PROGRAM Stn4
VAR

	start4: BOOL;
	reset4: BOOL;

	Stn4ProcessFE: F_TRIG;
	Stn4ProcessRE: R_TRIG;
	bCutStn4ProcessHalt: BOOL;
	DoorClose4: R_TRIG;
	bStn4DoorClamp: BOOL;
END_VAR
VAR // added by the converter: edge detectors and wires of the graphical bodies
    _w1, _w2 : ANY;
END_VAR

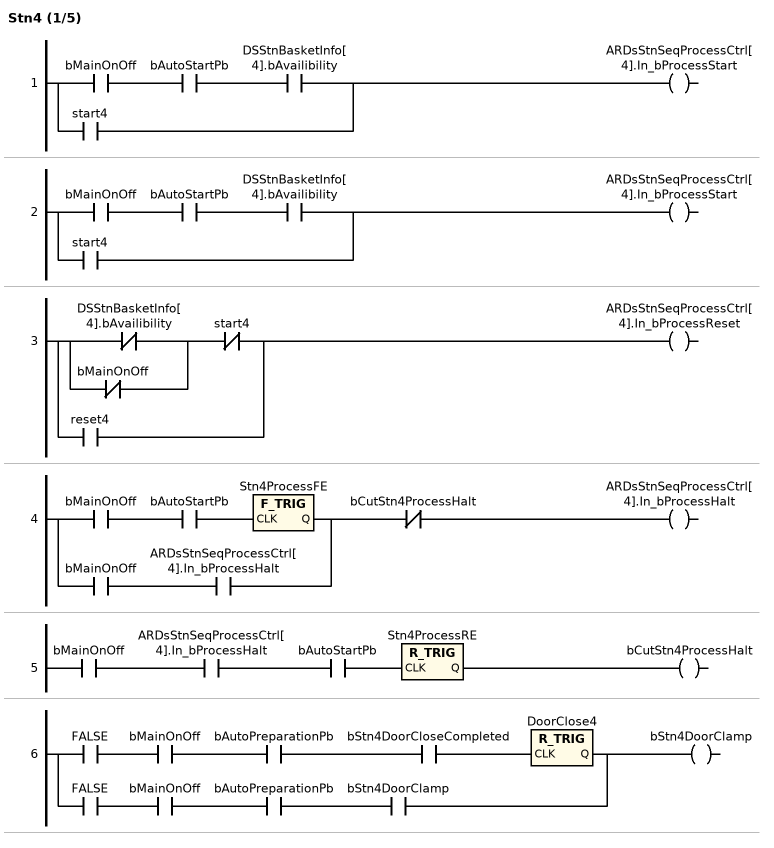
// NETWORK 1
ARDsStnSeqProcessCtrl[4].In_bProcessStart := bMainOnOff AND bAutoStartPb AND DSStnBasketInfo[4].bAvailibility OR start4;

// NETWORK 2
ARDsStnSeqProcessCtrl[4].In_bProcessStart := bMainOnOff AND bAutoStartPb AND DSStnBasketInfo[4].bAvailibility OR start4;

// NETWORK 3
ARDsStnSeqProcessCtrl[4].In_bProcessReset := (NOT DSStnBasketInfo[4].bAvailibility OR NOT bMainOnOff) AND NOT start4 OR reset4;

// NETWORK 4
Stn4ProcessFE(CLK := bMainOnOff AND bAutoStartPb); // F_TRIG
ARDsStnSeqProcessCtrl[4].In_bProcessHalt := (Stn4ProcessFE.Q OR bMainOnOff AND ARDsStnSeqProcessCtrl[4].In_bProcessHalt) AND NOT bCutStn4ProcessHalt;

// NETWORK 5
Stn4ProcessRE(CLK := bMainOnOff AND ARDsStnSeqProcessCtrl[4].In_bProcessHalt AND bAutoStartPb); // R_TRIG
bCutStn4ProcessHalt := Stn4ProcessRE.Q;

// NETWORK 6
DoorClose4(CLK := (FALSE AND bMainOnOff AND bAutoPreparationPb) AND bStn4DoorCloseCompleted); // R_TRIG
bStn4DoorClamp := DoorClose4.Q OR (FALSE AND bMainOnOff AND bAutoPreparationPb) AND bStn4DoorClamp;

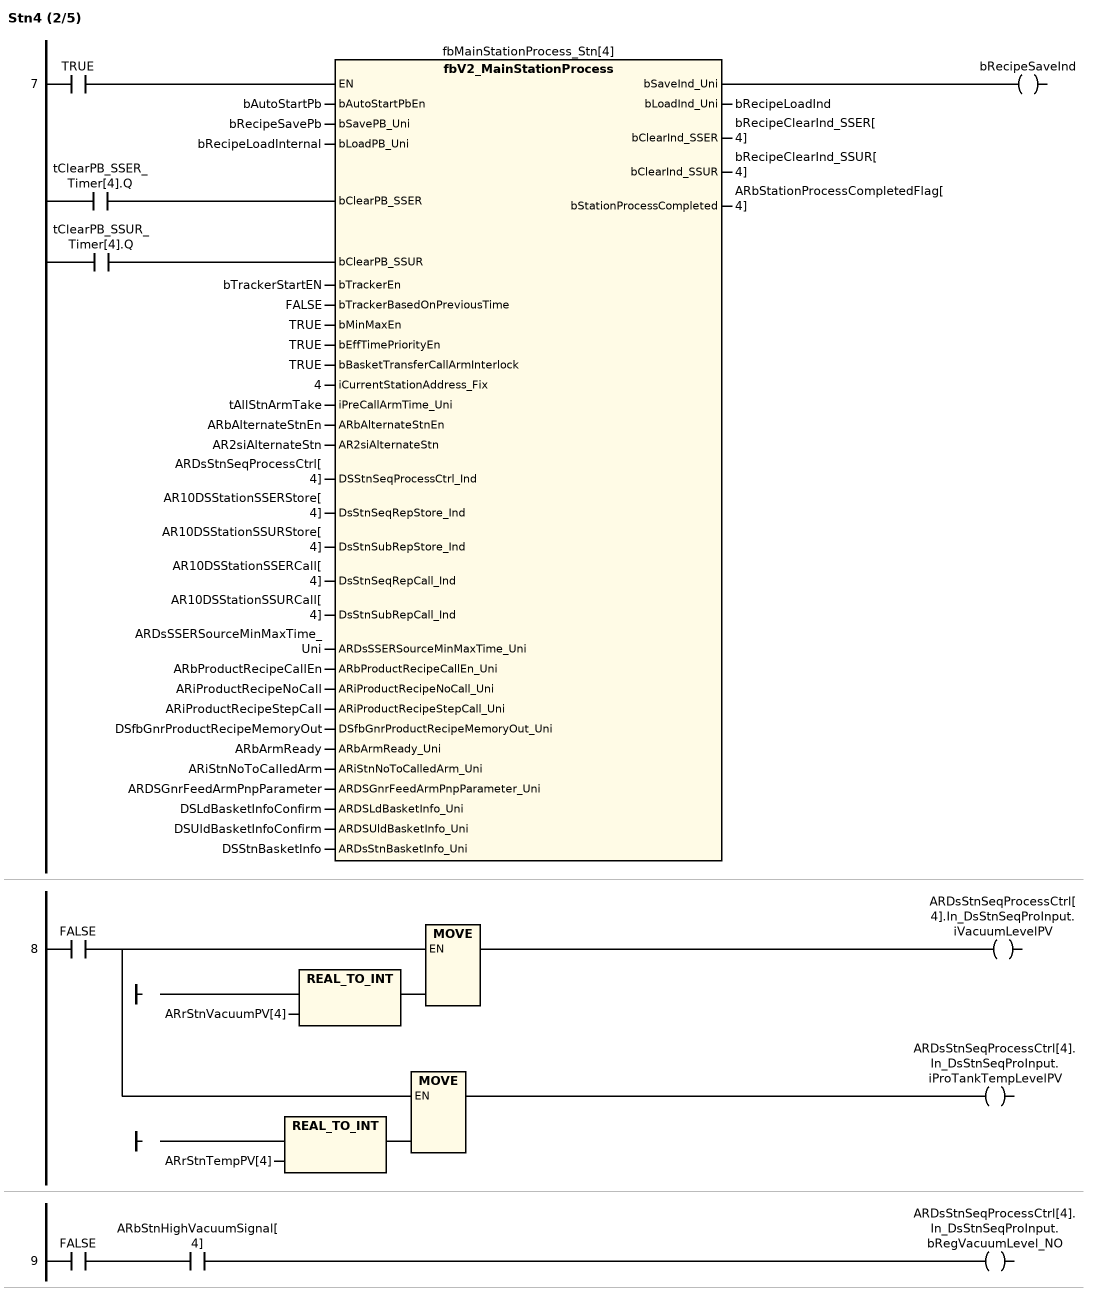
// NETWORK 7
fbMainStationProcess_Stn[4](
    bAutoStartPbEn := bAutoStartPb,
    bSavePB_Uni := bRecipeSavePb,
    bLoadPB_Uni := bRecipeLoadInternal,
    bClearPB_SSER := tClearPB_SSER_Timer[4].Q,
    bClearPB_SSUR := tClearPB_SSUR_Timer[4].Q,
    bTrackerEn := bTrackerStartEN,
    bTrackerBasedOnPreviousTime := FALSE,
    bMinMaxEn := TRUE,
    bEffTimePriorityEn := TRUE,
    bBasketTransferCallArmInterlock := TRUE,
    iCurrentStationAddress_Fix := 4,
    iPreCallArmTime_Uni := tAllStnArmTake,
    ARbAlternateStnEn := ARbAlternateStnEn,
    AR2siAlternateStn := AR2siAlternateStn,
    DSStnSeqProcessCtrl_Ind := ARDsStnSeqProcessCtrl[4],
    DsStnSeqRepStore_Ind := AR10DSStationSSERStore[4],
    DsStnSubRepStore_Ind := AR10DSStationSSURStore[4],
    DsStnSeqRepCall_Ind := AR10DSStationSSERCall[4],
    DsStnSubRepCall_Ind := AR10DSStationSSURCall[4],
    ARDsSSERSourceMinMaxTime_Uni := ARDsSSERSourceMinMaxTime_Uni,
    ARbProductRecipeCallEn_Uni := ARbProductRecipeCallEn,
    ARiProductRecipeNoCall_Uni := ARiProductRecipeNoCall,
    ARiProductRecipeStepCall_Uni := ARiProductRecipeStepCall,
    DSfbGnrProductRecipeMemoryOut_Uni := DSfbGnrProductRecipeMemoryOut,
    ARbArmReady_Uni := ARbArmReady,
    ARiStnNoToCalledArm_Uni := ARiStnNoToCalledArm,
    ARDSGnrFeedArmPnpParameter_Uni := ARDSGnrFeedArmPnpParameter,
    ARDSLdBasketInfo_Uni := DSLdBasketInfoConfirm,
    ARDSUldBasketInfo_Uni := DSUldBasketInfoConfirm,
    ARDsStnBasketInfo_Uni := DSStnBasketInfo,
    bLoadInd_Uni => bRecipeLoadInd,
    bClearInd_SSER => bRecipeClearInd_SSER[4],
    bClearInd_SSUR => bRecipeClearInd_SSUR[4],
    bStationProcessCompleted => ARbStationProcessCompletedFlag[4]); // fbV2_MainStationProcess
bRecipeSaveInd := fbMainStationProcess_Stn[4].bSaveInd_Uni;

// NETWORK 8
IF FALSE THEN _w1 := REAL_TO_INT(ARrStnVacuumPV[4]); END_IF
ARDsStnSeqProcessCtrl[4].In_DsStnSeqProInput.iVacuumLevelPV := _w1;
IF FALSE THEN _w2 := REAL_TO_INT(ARrStnTempPV[4]); END_IF
ARDsStnSeqProcessCtrl[4].In_DsStnSeqProInput.iProTankTempLevelPV := _w2;

// NETWORK 9
ARDsStnSeqProcessCtrl[4].In_DsStnSeqProInput.bRegVacuumLevel_NO := FALSE AND ARbStnHighVacuumSignal[4];

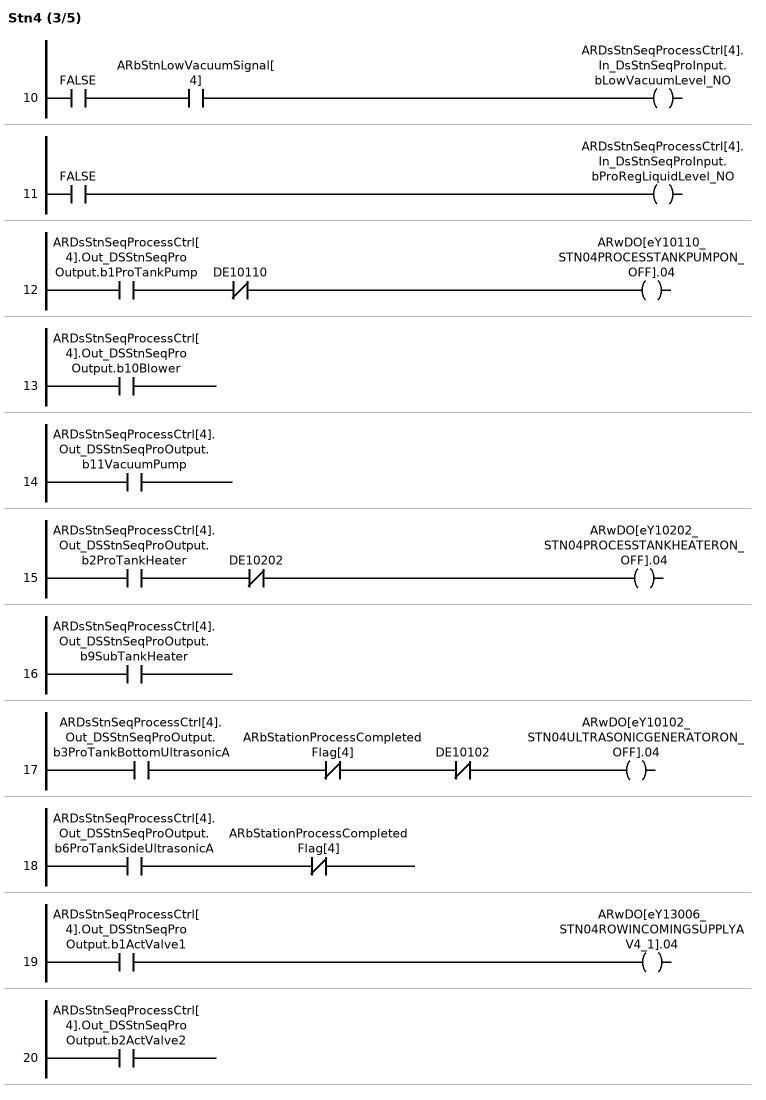
// NETWORK 10
ARDsStnSeqProcessCtrl[4].In_DsStnSeqProInput.bLowVacuumLevel_NO := FALSE AND ARbStnLowVacuumSignal[4];

// NETWORK 11
ARDsStnSeqProcessCtrl[4].In_DsStnSeqProInput.bProRegLiquidLevel_NO := FALSE;

// NETWORK 12
ARwDO[eY10110_STN04PROCESSTANKPUMPON_OFF].04 := ARDsStnSeqProcessCtrl[4].Out_DSStnSeqProOutput.b1ProTankPump AND NOT DE10110;

// NETWORK 13
(* ARDsStnSeqProcessCtrl[4].Out_DSStnSeqProOutput.b10Blower; not connected *)

// NETWORK 14
(* ARDsStnSeqProcessCtrl[4].Out_DSStnSeqProOutput.b11VacuumPump; not connected *)

// NETWORK 15
ARwDO[eY10202_STN04PROCESSTANKHEATERON_OFF].04 := ARDsStnSeqProcessCtrl[4].Out_DSStnSeqProOutput.b2ProTankHeater AND NOT DE10202;

// NETWORK 16
(* ARDsStnSeqProcessCtrl[4].Out_DSStnSeqProOutput.b9SubTankHeater; not connected *)

// NETWORK 17
ARwDO[eY10102_STN04ULTRASONICGENERATORON_OFF].04 := ARDsStnSeqProcessCtrl[4].Out_DSStnSeqProOutput.b3ProTankBottomUltrasonicA AND NOT ARbStationProcessCompletedFlag[4] AND NOT DE10102;

// NETWORK 18
(* ARDsStnSeqProcessCtrl[4].Out_DSStnSeqProOutput.b6ProTankSideUltrasonicA AND NOT ARbStationProcessCompletedFlag[4]; result not used *)

// NETWORK 19
ARwDO[eY13006_STN04ROWINCOMINGSUPPLYAV4_1].04 := ARDsStnSeqProcessCtrl[4].Out_DSStnSeqProOutput.b1ActValve1;

// NETWORK 20
(* ARDsStnSeqProcessCtrl[4].Out_DSStnSeqProOutput.b2ActValve2; not connected *)

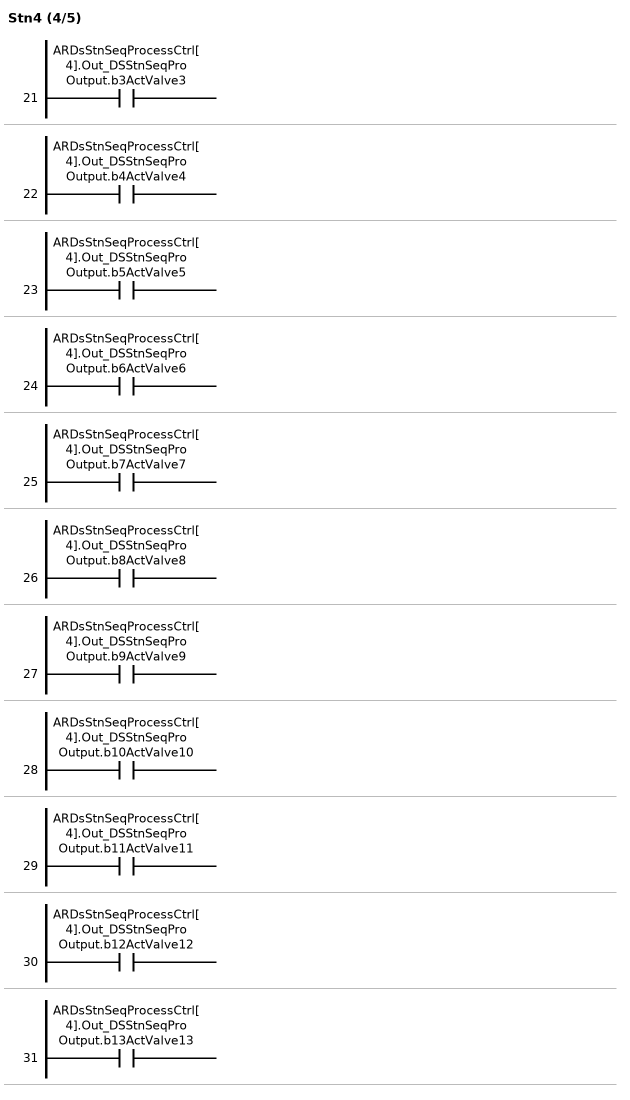
// NETWORK 21
(* ARDsStnSeqProcessCtrl[4].Out_DSStnSeqProOutput.b3ActValve3; not connected *)

// NETWORK 22
(* ARDsStnSeqProcessCtrl[4].Out_DSStnSeqProOutput.b4ActValve4; not connected *)

// NETWORK 23
(* ARDsStnSeqProcessCtrl[4].Out_DSStnSeqProOutput.b5ActValve5; not connected *)

// NETWORK 24
(* ARDsStnSeqProcessCtrl[4].Out_DSStnSeqProOutput.b6ActValve6; not connected *)

// NETWORK 25
(* ARDsStnSeqProcessCtrl[4].Out_DSStnSeqProOutput.b7ActValve7; not connected *)

// NETWORK 26
(* ARDsStnSeqProcessCtrl[4].Out_DSStnSeqProOutput.b8ActValve8; not connected *)

// NETWORK 27
(* ARDsStnSeqProcessCtrl[4].Out_DSStnSeqProOutput.b9ActValve9; not connected *)

// NETWORK 28
(* ARDsStnSeqProcessCtrl[4].Out_DSStnSeqProOutput.b10ActValve10; not connected *)

// NETWORK 29
(* ARDsStnSeqProcessCtrl[4].Out_DSStnSeqProOutput.b11ActValve11; not connected *)

// NETWORK 30
(* ARDsStnSeqProcessCtrl[4].Out_DSStnSeqProOutput.b12ActValve12; not connected *)

// NETWORK 31
(* ARDsStnSeqProcessCtrl[4].Out_DSStnSeqProOutput.b13ActValve13; not connected *)

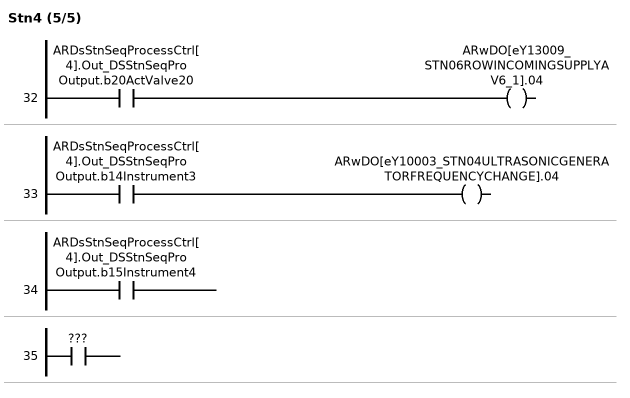
// NETWORK 32
ARwDO[eY13009_STN06ROWINCOMINGSUPPLYAV6_1].04 := ARDsStnSeqProcessCtrl[4].Out_DSStnSeqProOutput.b20ActValve20;

// NETWORK 33
ARwDO[eY10003_STN04ULTRASONICGENERATORFREQUENCYCHANGE].04 := ARDsStnSeqProcessCtrl[4].Out_DSStnSeqProOutput.b14Instrument3;

// NETWORK 34
(* ARDsStnSeqProcessCtrl[4].Out_DSStnSeqProOutput.b15Instrument4; not connected *)

// NETWORK 35

END_PROGRAM

(* stored: Version 1.1.0.1, ProductVersion 3.1.4024.12
   POU Stn4: Id {10afb006-1d86-4644-9731-7a04d5fe08a1}, SpecialFunc None *)
